FUNCTION F_SampleTimeCheck : BOOL
VAR_INPUT
	nSampleTimestamp: ULINT;
	nLastSampleTimestamp: ULINT;
	nSampleTime: UDINT;
END_VAR
VAR
	nDeviation: UDINT := 500000; //Allowed deviation 0.5ms
END_VAR

IF nLastSampleTimestamp = 0 THEN
	F_SampleTimeCheck:= TRUE;
ELSIF nSampleTimestamp >= (nLastSampleTimestamp + (nSampleTime + nDeviation)) THEN
	F_SampleTimeCheck:= TRUE;
ELSIF nSampleTimestamp >= (nLastSampleTimestamp + (nSampleTime - nDeviation)) THEN
	F_SampleTimeCheck:= TRUE;
ELSE
	F_SampleTimeCheck:= FALSE;
END_IF

END_FUNCTION

(* stored: POU F_SampleTimeCheck: Id 0faa84e9-754e-428d-ae6f-ebebaf33b37a, SpecialFunc None *)
